{attribute 'TcGenerated'}
// This function has been automatically generated from the project information.
VAR_GLOBAL CONSTANT
    {attribute 'const_non_replaced'}
    {attribute 'linkalways'}
    stLibVersion_SDS_M3 : ST_LibVersion := (iMajor := 1, iMinor := 1, iBuild := 0, iRevision := 0, sVersion := '1.1.0');
END_VAR

(* stored: Version 1.1.0.1, ProductVersion 3.1.4020.12
   GVL Global_Version: Id 154c2f9c-53a7-490a-b781-ea448d9f58a3 *)
